Yaskawa INFORM job: pneumatic_pod_cylinder_program.JBI

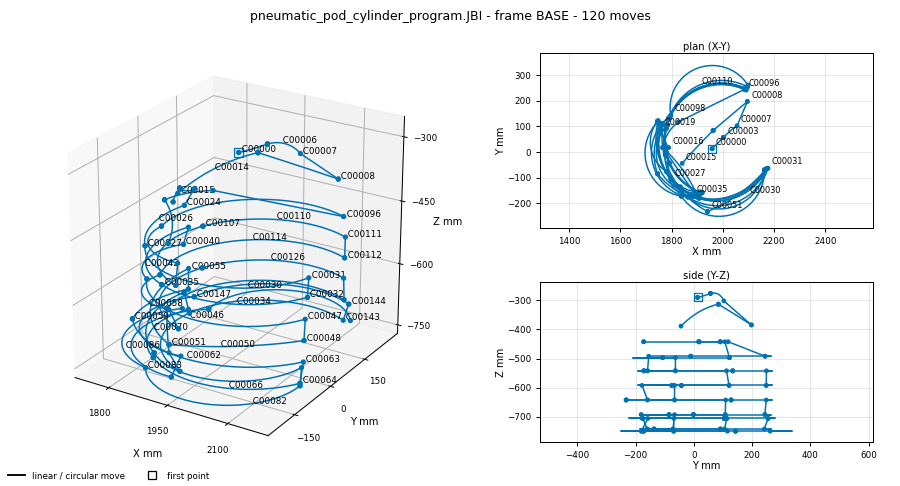
[picture p0: tool path of pneumatic_pod_cylinder_program.JBI in frame BASE, 120 of 166 moves have a stored position in this frame; points joined in program order, loops and branches not executed]
/JOB
//NAME pneumatic_pod_cylinder_program
//POS
///NPOS 160,0,160,0,0,0
///TOOL 0
///POSTYPE BASE
///RECTAN
///RCONF 0,0,0,0,0,0,0,0,0,0,0,0,0,0,0,0,0,0,0,0,0,0,0,0
C00000=1958.389235,12.976268,-289.886425,-175.000000,-11.803321,-5.000000
C00001=1958.389235,12.976268,-289.886425,-175.000000,-11.803321,-5.000000
C00002=1989.508045,44.082528,-281.112605,175.000000,-6.736144,5.000000
C00003=2002.234627,57.034265,-276.300191,173.720113,-5.000000,5.000000
C00004=2002.234627,57.034265,-276.300191,173.720113,-5.000000,5.000000
C00005=2002.234627,57.034265,-276.300191,173.720113,-5.000000,5.000000
C00006=2021.317158,75.250873,-275.482263,170.987178,-5.000000,5.000000
C00007=2055.940541,103.026667,-302.047678,165.858900,5.000000,-5.000000
C00008=2095.988887,197.429445,-384.323341,150.703461,15.702358,-8.634661
C00009=2095.988887,197.429445,-384.323341,150.703461,15.702358,-8.634661
C00010=2016.462182,130.189771,-341.598592,166.196837,5.000000,-5.000000
C00011=1962.352724,84.278253,-313.390552,174.835164,-5.875673,5.000000
C00012=1962.352724,84.278253,-313.390552,174.835164,-5.875673,5.000000
C00013=1962.352724,84.278253,-313.390552,174.835164,-5.875673,5.000000
C00014=1892.054622,12.128609,-343.204266,-171.950724,-18.467356,-5.000000
C00015=1841.583716,-44.157242,-388.454607,-157.126304,-26.974330,-10.833106
C00016=1787.842320,17.460255,-442.171500,-175.000000,-89.999999,5.000000
C00017=1787.842320,17.460255,-442.171500,-175.000000,-89.999999,5.000000
C00018=1762.763983,72.220182,-442.171500,168.173708,-90.000000,5.000000
C00019=1756.652008,90.892509,-442.171500,163.778025,-89.999999,5.000000
C00020=1756.652008,90.892509,-442.171500,163.778025,-89.999999,5.000000
C00021=1756.652008,90.892509,-442.171500,163.778025,-89.999999,5.000000
C00022=1785.884546,94.182511,-442.171500,160.453401,-90.000000,5.000000
C00023=1785.429307,106.503755,-442.171500,157.171649,-90.000000,5.000000
C00024=1747.586114,122.082867,-496.712000,157.422229,-89.999999,5.000000
C00025=1747.586114,122.082867,-496.712000,157.422229,-89.999999,5.000000
C00026=1742.596579,15.266334,-496.712000,-175.000000,-89.999999,5.000000
C00027=1798.217467,-107.210042,-496.712000,-141.599086,-89.999999,5.000000
C00028=1798.217467,-107.210042,-496.712000,-141.599086,-89.999999,5.000000
C00029=1798.217467,-107.210042,-496.712000,-141.599086,-89.999999,5.000000
C00030=2091.435568,-175.733861,-496.712000,-59.484566,-90.000000,5.000000
C00031=2176.600223,-63.140022,-496.712000,-24.179300,-90.000000,5.000000
C00032=2174.244974,-63.288750,-541.881500,-24.618751,-90.000000,5.000000
C00033=2174.244974,-63.288750,-541.881500,-24.618751,-90.000000,5.000000
C00034=2062.522244,-171.710489,-541.881500,-65.588851,-89.999999,5.000000
C00035=1882.924859,-171.618587,-541.881500,-113.630343,-90.000000,5.000000
C00036=1882.924859,-171.618587,-541.881500,-113.630343,-90.000000,5.000000
C00037=1882.924859,-171.618587,-541.881500,-113.630343,-90.000000,5.000000
C00038=1766.788315,-52.058745,-541.881500,-158.157674,-89.999999,5.000000
C00039=1764.709992,111.933306,-541.881500,158.300126,-90.000000,5.000000
C00040=1744.803569,120.918643,-591.866500,158.224242,-89.999999,5.000000
C00041=1744.803569,120.918643,-591.866500,158.224242,-89.999999,5.000000
C00042=1733.485377,-25.931279,-591.866500,-166.712945,-90.000000,5.000000
C00043=1779.551675,-75.626442,-591.866500,-151.122649,-90.000000,5.000000
C00044=1779.551675,-75.626442,-591.866500,-151.122649,-90.000000,5.000000
C00045=1779.551675,-75.626442,-591.866500,-151.122649,-90.000000,5.000000
C00046=1957.900310,-190.694442,-591.866500,-93.554499,-90.000000,5.000000
C00047=2171.194950,-66.216273,-591.866500,-25.811289,-89.999999,5.000000
C00048=2169.098166,-66.278490,-641.834500,-26.243734,-90.000000,5.000000
C00049=2169.098166,-66.278490,-641.834500,-26.243734,-90.000000,5.000000
C00050=2031.548258,-185.577959,-641.834500,-74.661465,-90.000000,5.000000
C00051=1940.438954,-232.092166,-641.834500,-96.888658,-90.000000,5.000000
C00052=1940.438954,-232.092166,-641.834500,-96.888658,-90.000000,5.000000
C00053=1940.438954,-232.092166,-641.834500,-96.888658,-90.000000,5.000000
C00054=1822.563016,-128.186854,-641.834500,-133.265491,-89.999999,5.000000
C00055=1765.603423,109.260868,-641.834500,159.202932,-90.000000,5.000000
C00056=1765.499466,107.658138,-692.401500,159.774109,-89.999999,5.000000
C00057=1765.499466,107.658138,-692.401500,159.774109,-89.999999,5.000000
C00058=1732.303208,-14.105595,-692.401500,-169.310028,-89.999999,5.000000
C00059=1745.517358,-85.170440,-692.401500,-152.867083,-89.999999,5.000000
C00060=1745.517358,-85.170440,-692.401500,-152.867083,-89.999999,5.000000
C00061=1745.517358,-85.170440,-692.401500,-152.867083,-89.999999,5.000000
C00062=1945.582904,-184.821395,-692.401500,-97.171938,-90.000000,5.000000
C00063=2167.950140,-66.166969,-692.401500,-26.534234,-89.999999,5.000000
C00064=2163.908798,-71.645912,-741.608000,-28.487004,-90.000000,5.000000
C00065=2163.908798,-71.645912,-741.608000,-28.487004,-90.000000,5.000000
C00066=2043.794149,-172.619930,-741.608000,-70.980234,-90.000000,5.000000
C00067=1834.088456,-136.294175,-741.608000,-129.643611,-90.000000,5.000000
C00068=1834.088456,-136.294175,-741.608000,-129.643611,-90.000000,5.000000
C00069=1834.088456,-136.294175,-741.608000,-129.643611,-90.000000,5.000000
C00070=1755.307009,-27.405749,-741.608000,-164.815329,-89.999999,5.000000
C00071=1766.265970,105.664864,-741.608000,160.360654,-89.999999,5.000000
C00072=1750.768421,112.897821,-705.313960,180.000000,-60.000000,-19.868150
C00073=1750.768421,112.897821,-705.313960,180.000000,-60.000000,-19.868150
C00074=1782.417120,-86.642602,-705.313960,-180.000000,-60.000000,31.836966
C00075=1863.483981,-175.594905,-705.313960,180.000000,-60.000000,62.019342
C00076=1863.483981,-175.594905,-705.313960,180.000000,-60.000000,62.019342
C00077=1863.483981,-175.594905,-705.313960,180.000000,-60.000000,62.019342
C00078=2099.334496,-182.161971,-705.313960,180.000000,-60.000000,120.324491
C00079=2165.317613,-68.688675,-705.313960,180.000000,-60.000000,152.192193
C00080=2162.402387,-69.212681,-749.043960,180.000000,-60.000000,151.539907
C00081=2162.402387,-69.212681,-749.043960,180.000000,-60.000000,151.539907
C00082=2115.752215,-193.881949,-749.043960,180.000000,-60.000000,121.956917
C00083=1838.164203,-172.427780,-749.043960,180.000000,-60.000000,56.405932
C00084=1838.164203,-172.427780,-749.043960,180.000000,-60.000000,56.405932
C00085=1838.164203,-172.427780,-749.043960,180.000000,-60.000000,56.405932
C00086=1742.022909,-120.019752,-749.043960,180.000000,-60.000000,33.309748
C00087=1743.750805,114.974889,-749.043960,180.000000,-60.000000,-19.633476
C00088=1901.594772,-172.069270,-442.010000,-113.547603,-90.000000,5.000000
C00089=1901.594772,-172.069270,-442.010000,-113.547603,-90.000000,5.000000
C00090=1830.042622,-51.785262,-442.010000,-149.794577,-90.000000,5.000000
C00091=1765.744080,17.324869,-442.010000,-173.171327,-90.000000,5.000000
C00092=1765.744080,17.324869,-442.010000,-173.171327,-90.000000,5.000000
C00093=1765.744080,17.324869,-442.010000,-173.171327,-90.000000,5.000000
C00094=1784.311178,69.500826,-442.010000,173.380676,-90.000000,5.000000
C00095=1826.843007,117.664577,-442.010000,156.748753,-90.000000,5.000000
C00096=2084.501148,244.731054,-491.806000,65.971125,-90.000000,5.000000
C00097=2084.501148,244.731054,-491.806000,65.971125,-90.000000,5.000000
C00098=1796.355608,144.183876,-491.806000,153.656022,-90.000000,5.000000
C00099=1775.580442,-10.759740,-491.806000,-165.664564,-90.000000,5.000000
C00100=1775.580442,-10.759740,-491.806000,-165.664564,-90.000000,5.000000
C00101=1775.580442,-10.759740,-491.806000,-165.664564,-90.000000,5.000000
C00102=1802.821395,-103.359707,-491.806000,-142.338297,-90.000000,5.000000
C00103=1913.008409,-154.827641,-491.806000,-112.424309,-90.000000,5.000000
C00104=1909.752136,-158.960265,-541.902000,-112.621130,-90.000000,5.000000
C00105=1909.752136,-158.960265,-541.902000,-112.621130,-90.000000,5.000000
C00106=1801.260468,-65.877178,-541.902000,-150.005655,-89.999999,5.000000
C00107=1789.016734,133.315309,-541.902000,157.059890,-90.000000,5.000000
C00108=1789.016734,133.315309,-541.902000,157.059890,-90.000000,5.000000
C00109=1789.016734,133.315309,-541.902000,157.059890,-90.000000,5.000000
C00110=1903.027306,249.788625,-541.902000,114.338832,-90.000000,5.000000
C00111=2087.842424,249.101612,-541.902000,65.470009,-90.000000,5.000000
C00112=2087.428895,248.291086,-591.876500,65.304442,-90.000000,5.000000
C00113=2087.428895,248.291086,-591.876500,65.304442,-90.000000,5.000000
C00114=1858.487770,221.794079,-591.876500,127.867986,-90.000000,5.000000
C00115=1791.184517,-42.628423,-591.876500,-156.318246,-90.000000,5.000000
C00116=1791.184517,-42.628423,-591.876500,-156.318246,-90.000000,5.000000
C00117=1791.184517,-42.628423,-591.876500,-156.318246,-90.000000,5.000000
C00118=1850.893373,-170.912390,-591.876500,-123.465716,-90.000000,5.000000
C00119=1904.579863,-177.863690,-591.876500,-111.871049,-90.000000,5.000000
C00120=1915.712840,-159.018102,-641.812500,-110.838420,-89.999999,5.000000
C00121=1915.712840,-159.018102,-641.812500,-110.838420,-89.999999,5.000000
C00122=1813.935599,-80.766240,-641.812500,-144.630892,-90.000000,5.000000
C00123=1789.735714,128.140997,-641.812500,158.403158,-90.000000,5.000000
C00124=1789.735714,128.140997,-641.812500,158.403158,-90.000000,5.000000
C00125=1789.735714,128.140997,-641.812500,158.403158,-90.000000,5.000000
C00126=1892.048580,242.435477,-641.812500,117.620654,-90.000000,5.000000
C00127=2086.001589,248.329483,-641.812500,65.468050,-90.000000,5.000000
C00128=2090.738990,243.748144,-691.879500,63.661386,-90.000000,5.000000
C00129=2090.738990,243.748144,-691.879500,63.661386,-90.000000,5.000000
C00130=1878.366227,233.035654,-691.879500,121.907299,-89.999999,5.000000
C00131=1780.077467,-1.553944,-691.879500,-166.999496,-89.999999,5.000000
C00132=1780.077467,-1.553944,-691.879500,-166.999496,-89.999999,5.000000
C00133=1780.077467,-1.553944,-691.879500,-166.999496,-89.999999,5.000000
C00134=1873.587340,-137.072387,-691.879500,-123.019771,-90.000000,5.000000
C00135=1905.371037,-180.759490,-691.879500,-111.135559,-90.000000,5.000000
C00136=1918.425883,-159.724483,-741.677500,-109.774762,-90.000000,5.000000
C00137=1918.425883,-159.724483,-741.677500,-109.774762,-90.000000,5.000000
C00138=1820.827034,-87.730870,-741.677500,-141.717513,-89.999999,5.000000
C00139=1778.635674,91.138930,-741.677500,168.720641,-89.999999,5.000000
C00140=1778.635674,91.138930,-741.677500,168.720641,-89.999999,5.000000
C00141=1778.635674,91.138930,-741.677500,168.720641,-89.999999,5.000000
C00142=1869.340799,227.532997,-741.677500,124.658787,-90.000000,5.000000
C00143=2090.708893,241.748945,-741.677500,63.251785,-90.000000,5.000000
C00144=2096.916105,254.617328,-705.374460,180.000000,-60.000000,-116.859702
C00145=2096.916105,254.617328,-705.374460,180.000000,-60.000000,-116.859702
C00146=1860.446002,232.248402,-705.374460,-180.000000,-60.000000,-54.186178
C00147=1783.326484,104.169568,-705.374460,-180.000000,-60.000000,-14.781315
C00148=1783.326484,104.169568,-705.374460,-180.000000,-60.000000,-14.781315
C00149=1783.326484,104.169568,-705.374460,-180.000000,-60.000000,-14.781315
C00150=1785.330126,-113.298118,-705.374460,180.000000,-60.000000,38.028554
C00151=1920.424328,-158.163432,-705.374460,180.000000,-60.000000,70.750091
C00152=1909.690689,-179.845646,-748.994960,-180.000000,-60.000000,70.181437
C00153=1909.690689,-179.845646,-748.994960,-180.000000,-60.000000,70.181437
C00154=1777.431556,-131.990829,-748.994960,180.000000,-60.000000,40.171089
C00155=1796.968246,142.908579,-748.994960,180.000000,-60.000000,-25.577010
C00156=1796.968246,142.908579,-748.994960,180.000000,-60.000000,-25.577010
C00157=1796.968246,142.908579,-748.994960,180.000000,-60.000000,-25.577010
C00158=1831.061727,277.162062,-748.994960,180.000000,-60.000000,-54.700941
C00159=2097.945493,262.000831,-748.994960,-180.000000,-60.000000,-116.422269
///POSTYPE PULSE
///PULSE
EX00000=0
EX00001=92160
EX00002=184320
EX00003=276480
///POSTYPE PULSE
///PULSE
EC00000=0
EC00001=0
EC00002=0
EC00003=0
EC00004=0
EC00005=0
EC00006=0
EC00007=0
EC00008=0
EC00009=0
EC00010=0
EC00011=0
EC00012=0
EC00013=0
EC00014=0
EC00015=0
EC00016=184320
EC00017=184320
EC00018=184320
EC00019=184320
EC00020=184320
EC00021=184320
EC00022=184320
EC00023=184320
EC00024=184320
EC00025=184320
EC00026=184320
EC00027=184320
EC00028=184320
EC00029=184320
EC00030=184320
EC00031=184320
EC00032=184320
EC00033=184320
EC00034=184320
EC00035=184320
EC00036=184320
EC00037=184320
EC00038=184320
EC00039=184320
EC00040=184320
EC00041=184320
EC00042=184320
EC00043=184320
EC00044=184320
EC00045=184320
EC00046=184320
EC00047=184320
EC00048=184320
EC00049=184320
EC00050=184320
EC00051=184320
EC00052=184320
EC00053=184320
EC00054=184320
EC00055=184320
EC00056=184320
EC00057=184320
EC00058=184320
EC00059=184320
EC00060=184320
EC00061=184320
EC00062=184320
EC00063=184320
EC00064=184320
EC00065=184320
EC00066=184320
EC00067=184320
EC00068=184320
EC00069=184320
EC00070=184320
EC00071=184320
EC00072=184320
EC00073=184320
EC00074=184320
EC00075=184320
EC00076=184320
EC00077=184320
EC00078=184320
EC00079=184320
EC00080=184320
EC00081=184320
EC00082=184320
EC00083=184320
EC00084=184320
EC00085=184320
EC00086=184320
EC00087=184320
EC00088=276480
EC00089=276480
EC00090=276480
EC00091=276480
EC00092=276480
EC00093=276480
EC00094=276480
EC00095=276480
EC00096=276480
EC00097=276480
EC00098=276480
EC00099=276480
EC00100=276480
EC00101=276480
EC00102=276480
EC00103=276480
EC00104=276480
EC00105=276480
EC00106=276480
EC00107=276480
EC00108=276480
EC00109=276480
EC00110=276480
EC00111=276480
EC00112=276480
EC00113=276480
EC00114=276480
EC00115=276480
EC00116=276480
EC00117=276480
EC00118=276480
EC00119=276480
EC00120=276480
EC00121=276480
EC00122=276480
EC00123=276480
EC00124=276480
EC00125=276480
EC00126=276480
EC00127=276480
EC00128=276480
EC00129=276480
EC00130=276480
EC00131=276480
EC00132=276480
EC00133=276480
EC00134=276480
EC00135=276480
EC00136=276480
EC00137=276480
EC00138=276480
EC00139=276480
EC00140=276480
EC00141=276480
EC00142=276480
EC00143=276480
EC00144=276480
EC00145=276480
EC00146=276480
EC00147=276480
EC00148=276480
EC00149=276480
EC00150=276480
EC00151=276480
EC00152=276480
EC00153=276480
EC00154=276480
EC00155=276480
EC00156=276480
EC00157=276480
EC00158=276480
EC00159=276480
//INST
///DATE 2023/08/07 13:43
///ATTR SC,RW,RJ
////FRAME BASE
///GROUP1 RB1,ST1
NOP
MOVJ P009 EX000 VJ=15.00
MOVJ C00000 EC00000 VJ=15.0
CALL JOB:SPYON
MOVC C00001 EC00001 V=150.0
MOVC C00002 EC00002 V=150.0
MOVC C00003 EC00003 V=150.0
MOVL C00004 EC00004 V=150.0
MOVC C00005 EC00005 V=150.0
MOVC C00006 EC00006 V=150.0
MOVC C00007 EC00007 V=150.0
MOVL C00008 EC00008 V=150.0
MOVC C00009 EC00009 V=150.0
MOVC C00010 EC00010 V=150.0
MOVC C00011 EC00011 V=150.0
MOVL C00012 EC00012 V=150.0
MOVC C00013 EC00013 V=150.0
MOVC C00014 EC00014 V=150.0
MOVC C00015 EC00015 V=150.0
CALL JOB:SPYOF
MOVJ P009 VJ=15.00
MOVJ P009 VJ=15.00
MOVJ P009 VJ=15.00
MOVJ C00016 EC00016 VJ=15.0
CALL JOB:SPYON
MOVC C00017 EC00017 V=150.0
MOVC C00018 EC00018 V=150.0
MOVC C00019 EC00019 V=150.0
MOVL C00020 EC00020 V=150.0
MOVC C00021 EC00021 V=150.0
MOVC C00022 EC00022 V=150.0
MOVC C00023 EC00023 V=150.0
MOVL C00024 EC00024 V=150.0
MOVC C00025 EC00025 V=150.0
MOVC C00026 EC00026 V=150.0
MOVC C00027 EC00027 V=150.0
MOVL C00028 EC00028 V=150.0
MOVC C00029 EC00029 V=150.0
MOVC C00030 EC00030 V=150.0
MOVC C00031 EC00031 V=150.0
MOVL C00032 EC00032 V=150.0
MOVC C00033 EC00033 V=150.0
MOVC C00034 EC00034 V=150.0
MOVC C00035 EC00035 V=150.0
MOVL C00036 EC00036 V=150.0
MOVC C00037 EC00037 V=150.0
MOVC C00038 EC00038 V=150.0
MOVC C00039 EC00039 V=150.0
MOVL C00040 EC00040 V=150.0
MOVC C00041 EC00041 V=150.0
MOVC C00042 EC00042 V=150.0
MOVC C00043 EC00043 V=150.0
MOVL C00044 EC00044 V=150.0
MOVC C00045 EC00045 V=150.0
MOVC C00046 EC00046 V=150.0
MOVC C00047 EC00047 V=150.0
MOVL C00048 EC00048 V=150.0
MOVC C00049 EC00049 V=150.0
MOVC C00050 EC00050 V=150.0
MOVC C00051 EC00051 V=150.0
MOVL C00052 EC00052 V=150.0
MOVC C00053 EC00053 V=150.0
MOVC C00054 EC00054 V=150.0
MOVC C00055 EC00055 V=150.0
MOVL C00056 EC00056 V=150.0
MOVC C00057 EC00057 V=150.0
MOVC C00058 EC00058 V=150.0
MOVC C00059 EC00059 V=150.0
MOVL C00060 EC00060 V=150.0
MOVC C00061 EC00061 V=150.0
MOVC C00062 EC00062 V=150.0
MOVC C00063 EC00063 V=150.0
MOVL C00064 EC00064 V=150.0
MOVC C00065 EC00065 V=150.0
MOVC C00066 EC00066 V=150.0
MOVC C00067 EC00067 V=150.0
MOVL C00068 EC00068 V=150.0
MOVC C00069 EC00069 V=150.0
MOVC C00070 EC00070 V=150.0
MOVC C00071 EC00071 V=150.0
MOVL C00072 EC00072 V=150.0
MOVC C00073 EC00073 V=150.0
MOVC C00074 EC00074 V=150.0
MOVC C00075 EC00075 V=150.0
MOVL C00076 EC00076 V=150.0
MOVC C00077 EC00077 V=150.0
MOVC C00078 EC00078 V=150.0
MOVC C00079 EC00079 V=150.0
MOVL C00080 EC00080 V=150.0
MOVC C00081 EC00081 V=150.0
MOVC C00082 EC00082 V=150.0
MOVC C00083 EC00083 V=150.0
MOVL C00084 EC00084 V=150.0
MOVC C00085 EC00085 V=150.0
MOVC C00086 EC00086 V=150.0
MOVC C00087 EC00087 V=150.0
CALL JOB:SPYOF
MOVJ P009 VJ=15.00
MOVJ C00088 EC00088 VJ=15.0
CALL JOB:SPYON
MOVC C00089 EC00089 V=150.0
MOVC C00090 EC00090 V=150.0
MOVC C00091 EC00091 V=150.0
MOVL C00092 EC00092 V=150.0
MOVC C00093 EC00093 V=150.0
MOVC C00094 EC00094 V=150.0
MOVC C00095 EC00095 V=150.0
MOVL C00096 EC00096 V=150.0
MOVC C00097 EC00097 V=150.0
MOVC C00098 EC00098 V=150.0
MOVC C00099 EC00099 V=150.0
MOVL C00100 EC00100 V=150.0
MOVC C00101 EC00101 V=150.0
MOVC C00102 EC00102 V=150.0
MOVC C00103 EC00103 V=150.0
MOVL C00104 EC00104 V=150.0
MOVC C00105 EC00105 V=150.0
MOVC C00106 EC00106 V=150.0
MOVC C00107 EC00107 V=150.0
MOVL C00108 EC00108 V=150.0
MOVC C00109 EC00109 V=150.0
MOVC C00110 EC00110 V=150.0
MOVC C00111 EC00111 V=150.0
MOVL C00112 EC00112 V=150.0
MOVC C00113 EC00113 V=150.0
MOVC C00114 EC00114 V=150.0
MOVC C00115 EC00115 V=150.0
MOVL C00116 EC00116 V=150.0
MOVC C00117 EC00117 V=150.0
MOVC C00118 EC00118 V=150.0
MOVC C00119 EC00119 V=150.0
MOVL C00120 EC00120 V=150.0
MOVC C00121 EC00121 V=150.0
MOVC C00122 EC00122 V=150.0
MOVC C00123 EC00123 V=150.0
MOVL C00124 EC00124 V=150.0
MOVC C00125 EC00125 V=150.0
MOVC C00126 EC00126 V=150.0
MOVC C00127 EC00127 V=150.0
MOVL C00128 EC00128 V=150.0
MOVC C00129 EC00129 V=150.0
MOVC C00130 EC00130 V=150.0
MOVC C00131 EC00131 V=150.0
MOVL C00132 EC00132 V=150.0
MOVC C00133 EC00133 V=150.0
MOVC C00134 EC00134 V=150.0
MOVC C00135 EC00135 V=150.0
MOVL C00136 EC00136 V=150.0
MOVC C00137 EC00137 V=150.0
MOVC C00138 EC00138 V=150.0
MOVC C00139 EC00139 V=150.0
MOVL C00140 EC00140 V=150.0
MOVC C00141 EC00141 V=150.0
MOVC C00142 EC00142 V=150.0
MOVC C00143 EC00143 V=150.0
MOVL C00144 EC00144 V=150.0
MOVC C00145 EC00145 V=150.0
MOVC C00146 EC00146 V=150.0
MOVC C00147 EC00147 V=150.0
MOVL C00148 EC00148 V=150.0
MOVC C00149 EC00149 V=150.0
MOVC C00150 EC00150 V=150.0
MOVC C00151 EC00151 V=150.0
MOVL C00152 EC00152 V=150.0
MOVC C00153 EC00153 V=150.0
MOVC C00154 EC00154 V=150.0
MOVC C00155 EC00155 V=150.0
MOVL C00156 EC00156 V=150.0
MOVC C00157 EC00157 V=150.0
MOVC C00158 EC00158 V=150.0
MOVC C00159 EC00159 V=150.0
CALL JOB:SPYOF
MOVJ P009 VJ=15.00
END
